FUNCTION_BLOCK PUBLIC PAERotationControl EXTENDS PAESensorDigital
VAR_INPUT
END_VAR
VAR_OUTPUT
END_VAR
VAR
	_SignalIsImpulse : BOOL;
END_VAR

METHOD FB_postinit
VAR_INPUT
	root : IACVariobatch;
END_VAR
SUPER^.FB_postinit(root);
root.OnPropertyChangedBool(THIS^, 36, _SignalIsImpulse);
END_METHOD

METHOD PUBLIC InvokeSetterBool
VAR_INPUT
	PropertyID : INT;
	PropertyValue : BOOL;
END_VAR
SUPER^.InvokeSetterBool(PropertyID, PropertyValue);
IF PropertyID = 36 THEN
	SignalIsImpulse := PropertyValue;
END_IF
END_METHOD

METHOD OnInitMemory
VAR_INPUT
	root : IACVariobatch;
END_VAR
RegisterProperty(root, 36, GCL.cSizeBYTE); //SignalIsImpulse
SUPER^.OnInitMemory(root);
END_METHOD

{attribute 'monitoring' := 'call'}
//{attribute 'TcRpcEnable'}
PROPERTY PUBLIC SignalIsImpulse : BOOL
GET // PUBLIC
SignalIsImpulse := _SignalIsImpulse;
END_GET
SET // PUBLIC
_SignalIsImpulse := SignalIsImpulse;
Root.OnPropertyChangedBool(THIS^, 36, _SignalIsImpulse);
END_SET
END_PROPERTY

END_FUNCTION_BLOCK

(* stored: Version 1.1.0.1, ProductVersion 3.1.4024.6
   POU PAERotationControl: Id {84bf60f1-2966-478d-a948-ae21a0430704}, SpecialFunc None
   Method FB_postinit: Id {07681089-ed89-4e22-ab59-77968c6433ea}
   Method InvokeSetterBool: Id {14e10b05-17a0-4858-a1a2-e191546db07a}
   Method OnInitMemory: Id {f8e08591-2f20-4557-8fda-98aedea31809}
   Property SignalIsImpulse: Id {7251a4c7-52f9-46c8-91cd-4393fcbd4979}
   Get Get: Id {974f5c70-5cf4-46fe-97fe-979891477eb7}
   Set Set: Id {950df7db-b8a5-440f-83ef-56eac21587c9} *)
